TYPE Vec2d : ARRAY[1..2] OF LREAL; END_TYPE

(* stored: Version 1.1.0.1, ProductVersion 3.1.4024.12
   DUT Vec2d: Id {f5244a8a-0c28-4681-aa4b-e8c56a89cbe6} *)
